// TIA Portal V19 export
DATA_BLOCK "AccRollConveyor"   // DB154
// stored: InstanceOfName AccRollConveyor_FB, InstanceOfType FB
"AccRollConveyor_FB"
   // VAR_INPUT
   //    AreaInterface : "AreaInterface";
   //    ZSI : "udt_ZoneSafetyInterface";
   //    DSI : Struct
   //       Roll1 : "udt_DeviceSafetyInterface";
   //       Roll2 : "udt_DeviceSafetyInterface";
   //       Roll3 : "udt_DeviceSafetyInterface";
   //       PusherVert : "udt_DeviceSafetyInterface";
   //       PusherHoriz : "udt_DeviceSafetyInterface";
   //    END_STRUCT;
   //    Drive : Struct
   //       Roll1 : "TAx_DriveInterface";
   //       Roll2 : "TAx_DriveInterface";
   //       Roll3 : "TAx_DriveInterface";
   //    END_STRUCT;
   //    HWID : Struct
   //       Roll1_TEL1 : HW_SUBMODULE;
   //       Roll2_TEL1 : HW_SUBMODULE;
   //       Roll3_TEL1 : HW_SUBMODULE;
   //    END_STRUCT;
   //    DataIn : Struct
   //       Pb_Semiauto : Bool;
   //       Rolls_PbFwd : Bool;
   //       Rolls_PbBwd : Bool;
   //       PusherVert_PbUp : Bool;
   //       PusherVert_PbDown : Bool;
   //       PusherHoriz_PbLeft : Bool;
   //       PusherHoriz_PbRight : Bool;
   //       SensorMatPresence_S2_Entry : Bool;
   //       SensorMatPresence_S3 : Bool;
   //       SensorMatPresence_S4 : Bool;
   //       SensorMatPresence_S5_Stop : Bool;
   //       ExitLeft_MatPresence1 : Bool;
   //       ExitLeft_MatPresence2 : Bool;
   //       ExitLeft_MatPresence3 : Bool;
   //       ExitLeft_MatPresence4 : Bool;
   //    END_STRUCT;
   //    CIn : Struct
   //       Manager : Struct
   //          EnableStopDoorOpeningReq : Bool;
   //          EnableStopInPhase : Bool;
   //          EnableStopProgrammed : Bool;
   //       END_STRUCT;
   //       Semiautomatic : Bool;
   //       A03_CanLoadPiece : Bool;
   //       A03_InCycle : Bool;
   //       ReqFwdFromCut : Bool;
   //       StopCheckQuality : Bool;
   //    END_STRUCT;
   //    Config : Struct
   //       Roll1 : "SpeedMachine_Config";
   //       Roll2 : "SpeedMachine_Config";
   //       Roll3 : "SpeedMachine_Config";
   //       PusherVert : Array[1..6] of "ValveMachine_Config";
   //       PusherHoriz : Array[1..6] of "ValveMachine_Config";
   //       SensorsDelayOn : Time;
   //       SensorsDelayOff : Time;
   //       ExitLeftDelayOn : Time;
   //       ExitLeftDelayOff : Time;
   //    END_STRUCT;
   // END_VAR
   // VAR_OUTPUT
   //    MachineInterface : "MachineInterface";
   //    COut : Struct
   //       Rolls : Struct
   //          Infeed_ReqON : Bool;
   //          Bwd_CheckNext : Bool;
   //          Fwd_CheckNext : Bool;
   //          Standstill : Bool;
   //       END_STRUCT;
   //       PusherVert : Struct
   //          Rest_CheckNext : Bool;
   //          Work_CheckNext : Bool;
   //          AllStandstill : Bool;
   //          TwoUp : Bool;
   //          AllDown : Bool;
   //       END_STRUCT;
   //       PusherHoriz : Struct
   //          Left_CheckNext : Bool;
   //          Right_CheckNext : Bool;
   //          AllStandstill : Bool;
   //          InLeftPos : Bool;
   //          InRightPos : Bool;
   //       END_STRUCT;
   //       Manager : "udt_AccRollConveyor_COut_Manager";
   //    END_STRUCT;
   // END_VAR
   // VAR_IN_OUT
   //    Pers : "udt_AccRollConveyor_Pers";
   // END_VAR
   // VAR
   //    Sts : Struct
   //       Semiautomatic : Bool;
   //       OP_CanMoveFreely : Bool;
   //       NextTargetPathLeft : Bool;
   //       NextTargetPathRight : Bool;
   //       ActTargetPathLeft : Bool;
   //       ActTargetPathRight : Bool;
   //       TrkExitLeftFull : Bool;
   //       TrkPieceInRolls : Int;
   //       TrkPieceToCheckInRoll : Int;
   //       TrkPieceInLenght : LReal;
   //       TrkPieceRecondGoodFind : Int;
   //       StopCutCheckPiece : Bool;
   //       Pusher : Struct
   //          InLeftPos : Bool;
   //          InRightPos : Bool;
   //          UsedInLeftPos : Bool;
   //          UsedInRightPos : Bool;
   //          AllDown : Bool;
   //          TwoUp : Bool;
   //          Used : Array[1.."MAX_PUSHER"] of Bool;
   //       END_STRUCT;
   //       CycleTime : Struct
   //          PusherHoriz : Struct
   //             DT_W_Start : DTL;
   //             DT_W_Stop : DTL;
   //             DT_R_Start : DTL;
   //             DT_R_Stop : DTL;
   //             R_To_W_Exe : Bool;
   //             W_To_R_Exe : Bool;
   //             R_To_W_Items : Int;
   //             R_To_W_Sum : Time;
   //             W_To_R_Items : Int;
   //             W_To_R_Sum : Time;
   //          END_STRUCT;
   //          PPrf_PrgNoSave : DInt;
   //       END_STRUCT;
   //    END_STRUCT;
   //    Ctrl : Struct
   //       StopInPhase : Bool;
   //       StopProgrammed : Bool;
   //       Pb_Semiauto : Bool;
   //       Rolls : Struct
   //          Man_Fwd : Bool;
   //          Man_Bwd : Bool;
   //          Aut_SlowDown : Bool;
   //          Aut_Fwd : Bool;
   //          Vel : LReal;
   //          Entry_Vel : LReal;
   //          Acc : LReal;
   //          Dec : LReal;
   //       END_STRUCT;
   //       Pusher : Struct
   //          Man_Left : Bool;
   //          Man_Right : Bool;
   //          Man_Up : Bool;
   //          Man_Down : Bool;
   //          Aut_Left : Bool;
   //          Aut_Right : Bool;
   //          Aut_Up : Bool;
   //          Aut_Down : Bool;
   //       END_STRUCT;
   //       Cycle : Struct
   //          ReqNextMovePieceToLeft : Bool;
   //          ReqNextMovePieceToRight : Bool;
   //          ExeNextMovePieceToLeft : Bool;
   //          ExeNextMovePieceToRight : Bool;
   //          ReqMovePieceToLeft : Bool;
   //          ReqMovePieceToRight : Bool;
   //          ExeMovePieceToLeft : Bool;
   //          ExeMovePieceToRight : Bool;
   //       END_STRUCT;
   //    END_STRUCT;
   //    Alarm : Struct
   //       Roll1 : "SpeedMachine_Alr";
   //       Roll2 : "SpeedMachine_Alr";
   //       Roll3 : "SpeedMachine_Alr";
   //       PusherVert : Array[1.."MAX_PUSHER"] of "ValveAlr";
   //       PusherHoriz : Array[1.."MAX_PUSHER"] of "ValveAlr";
   //       TrkCloggedLeftExit : Bool;
   //       TrkCloggedRightA03 : Bool;
   //       TrkCloggedRollway : Bool;
   //       TrkWrongMismatch_P0 : Bool;
   //       TrkExitFullToChek : Bool;
   //    END_STRUCT;
   //    Warning : Struct
   //       Roll1 : "SpeedMachine_Wng";
   //       Roll2 : "SpeedMachine_Wng";
   //       Roll3 : "SpeedMachine_Wng";
   //       PusherVert : Array[1.."MAX_PUSHER"] of "ValveMachine_Wng";
   //       PusherHoriz : Array[1.."MAX_PUSHER"] of "ValveMachine_Wng";
   //    END_STRUCT;
   //    HMI : Struct
   //       PusherHoriz : Struct
   //          Last_R_to_W_ID : DInt;
   //          Last_R_to_W_Time : Time;
   //          Last_W_to_R_ID : DInt;
   //          Last_W_to_R_Time : Time;
   //          Avg_R_to_W_Time : Time;
   //          Avg_W_to_R_Time : Time;
   //          Avg_CycleTime_S : LReal;
   //          Buffer_R_to_W_Time : Array[1..10] of Struct
   //             ID : DInt;
   //             Value : Time;
   //          END_STRUCT;
   //          Buffer_W_to_R_Time : Array[1..10] of Struct
   //             ID : DInt;
   //             Value : Time;
   //          END_STRUCT;
   //       END_STRUCT;
   //    END_STRUCT;
   //    Roll1 : "SpeedMachine_FB";
   //    Roll2 : "SpeedMachine_FB";
   //    Roll3 : "SpeedMachine_FB";
   //    PusherVert : Array[1.."MAX_PUSHER"] of "ValveMachine_FB";
   //    PusherHoriz : Array[1.."MAX_PUSHER"] of "ValveMachine_FB";
   //    MatPresence_S2_Entry : "DelayOnOff_R";
   //    MatPresence_S3 : "DelayOnOff_R";
   //    MatPresence_S4 : "DelayOnOff_R";
   //    MatPresence_S5_Stop : "DelayOnOff_R";
   //    MatPresence_ExitLeft1 : "DelayOnOff_R";
   //    MatPresence_ExitLeft2 : "DelayOnOff_R";
   //    MatPresence_ExitLeft3 : "DelayOnOff_R";
   //    MatPresence_ExitLeft4 : "DelayOnOff_R";
   //    tonSlowDownRolls { S7_SetPoint := 'True'} : TON_TIME;
   //    tonStopRollformer : TON_TIME;
   //    tonSlowDownRollformer : TON_TIME;
   //    tonTrkMismatcP0 { S7_SetPoint := 'True'} : TON_TIME;
   //    Rollway_Control : "Rulliera_Control_FB";
   //    AUX : Struct
   //       Pb_Semiauto { ExternalAccessible := 'False'; ExternalVisible := 'False'; ExternalWritable := 'False'} : Bool;
   //       Rolls_PbFwd : Bool;
   //       Rolls_PbBwd : Bool;
   //       PusherVert_PbUp : Bool;
   //       PusherVert_PbDopwn : Bool;
   //       PusherHoriz_PbLeft : Bool;
   //       PusherHoriz_PbRight : Bool;
   //       NE_MatPresence2_Entry { ExternalAccessible := 'False'; ExternalVisible := 'False'; ExternalWritable := 'False'} : Bool;
   //       PE_MatPresence3 : Bool;
   //       PE_MatPresence5_Stop : Bool;
   //       PE_SlowDownRolls : Bool;
   //       NE_SlowDownDone : Bool;
   //       PusherHoriz_InLeftPos : Bool;
   //       PusherHoriz_InRightPos : Bool;
   //    END_STRUCT;
   //    PusherVert_MachineInterface { ExternalAccessible := 'False'; ExternalVisible := 'False'; ExternalWritable := 'False'} : "MachineInterface";
   //    PusherHoriz_MachineInterface { ExternalAccessible := 'False'; ExternalVisible := 'False'; ExternalWritable := 'False'} : "MachineInterface";
   // END_VAR
BEGIN
   AreaInterface.EStop := FALSE;
   AreaInterface.Man := TRUE;
   AreaInterface.Aut := FALSE;
   AreaInterface.Cycle := FALSE;
   AreaInterface.StopInPhase := FALSE;
   AreaInterface.StopProgrammed := FALSE;
   AreaInterface.RstAlarms := FALSE;
   AreaInterface.ManOneShot := FALSE;
   AreaInterface.AutOneShot := FALSE;
   AreaInterface.CycleOneShot := FALSE;
   AreaInterface.CheckAutReady := FALSE;
   MachineInterface.AutReady := FALSE;
   MachineInterface.Aborting := FALSE;
   MachineInterface.AckStopInPhase := FALSE;
   MachineInterface.AckStopProgrammed := FALSE;
   MachineInterface.MotionsStandStill := TRUE;
   MachineInterface.AlarmsPresence := FALSE;
   MachineInterface.WarningPresence := FALSE;
END_DATA_BLOCK
